PROGRAM P_MyLight_Test_ST
VAR
	fbMyLight			:	FB_MyLight;
	bOn					:	BOOL;
	bOff				:	BOOL;
	bRecallMinLevel		:	BOOL;
	bSetControlLevel	:	BOOL;
	nSetControlLevel	:	BYTE;
	bControlLevel		:	BOOL;
	nControlLevel		:	BYTE;
END_VAR

fbMyLight();

IF (bOn) THEN
	fbMyLight.M_On();
	bOn := FALSE;
END_IF
IF (bOff) THEN
	fbMyLight.M_Off();
	bOff := FALSE;
END_IF
IF (bRecallMinLevel) THEN
	fbMyLight.M_RecallMinLevel();
	bRecallMinLevel := FALSE;
END_IF
IF (bSetControlLevel) THEN
	fbMyLight.M_SetControlLevel(nSetControlLevel);
	bSetControlLevel := FALSE;
END_IF

bControlLevel := fbMyLight.bControlLevel;
nControlLevel := fbMyLight.nControlLevel;

END_PROGRAM

(* stored: Version 1.1.0.1, ProductVersion 3.1.4024.12
   POU P_MyLight_Test_ST: Id {8d5c2de6-c612-4a36-8f71-3b8183571ca3}, SpecialFunc None *)
